// TIA Portal V20 export
DATA_BLOCK "SBK03"   // DB216
// stored: MemoryReserve 100
   VAR
      "X1-0 Roll change LH: Auto" : Bool;
      "X2-1 Roll change RH: Auto" : Bool;
      "X3-2 CART Detect Sensor 1" : Bool;
      "X4-3 CART Detect Sensor 2" : Bool;
      "X1-4 Roll change LH: Change" : Bool;
      "X2-5 Roll change RH: Change" : Bool;
      "X3-6 reserved" : Bool;
      "X4-7 reserved" : Bool;
      "X5-0 Roll change LH: Roll change in progress" : Bool;
      "X6-1 Roll change RH: Roll change in progress" : Bool;
      "X7-2 reserved" : Bool;
   END_VAR
BEGIN
END_DATA_BLOCK
